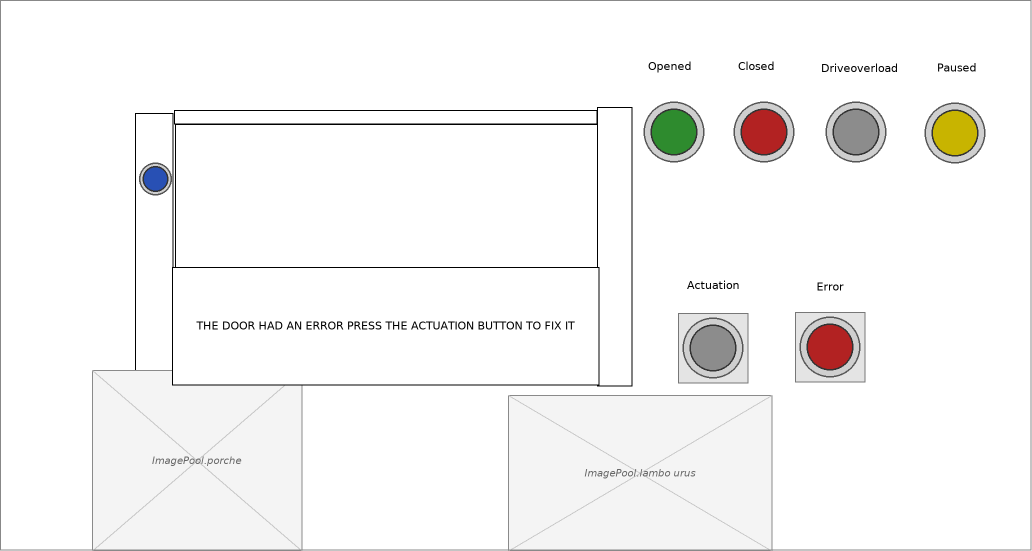
VISUALIZATION Visualization  // 1032x551
    Rectangle (175,124 424x261), invisible if: GarageDoor.bOpenSensor
    Rectangle (135,113 38x274)
    Rectangle (597,107 35x279)
    Rectangle (174,110 423x14)
    Lamp1 (136,160 39x38), variable: GarageDoor.bLightForMotion, style: Lamp-Lamp1-Blue
    Lamp1 (639,97 70x70), variable: GarageDoor.bOpenSensor, style: Lamp-Lamp1-Green
    Lamp1 (729,97 70x70), variable: GarageDoor.bClosedSensor, style: Lamp-Lamp1-Red
    Lamp1 (821,97 70x70), variable: GarageDoor.bDriveOverloadSensor, style: Lamp-Lamp1-Gray
    Label (637,52 66x29), "Opened"
    Label (730,55 53x23), "Closed"
    Label (816,57 87x23), "Driveoverload"
    PushSwitch (678,313 70x70), variable: GarageDoor.bActuationButton, behaviour: TAP, style: Switch-PushSwitch-Gray
    PushSwitch (795,312 70x70), variable: GarageDoor.bErrorButton, behaviour: TAP, style: Switch-PushSwitch-Red
    Label (804,263 52x48), "Error"
    Label (688,268 51x35), "Actuation"
    Lamp1 (920,98 70x70), variable: GarageDoor.bPauseLight, style: Lamp-Lamp1-Yellow
    Label (882,53 150x30), "Paused"
    Image (92,370 210x181), image: ImagePool.porche
    Image (508,395 264x156), image: ImagePool.lambo urus
    Rectangle (175,267 422x118), invisible if: NOT GarageDoor.bVisualizationOpenClose
    Rectangle (172,267 427x118), "THE DOOR HAD AN ERROR PRESS THE ACTUATION BUTTON TO FIX IT", invisible if: NOT GarageDoor.bDriveOverloadSensor
END_VISUALIZATION

(* stored: Version 1.1.0.1, ProductVersion 3.1.4024.12
   Visu Visualization: Id {9bae951d-5bd3-4968-ad88-f9e5223ad017} *)
